(* CoDeSys 2.3 library: TcSystemCX.lib *)
(* Libraries: STANDARD.LIB 5.6.98 12:03:02, TcBase.lib*14.5.09 12:14:08, TcSystem.lib*21.1.15 10:22:54 *)

(* Global variable list: Global_Constants *)
VAR_GLOBAL CONSTANT
	iLength						 : INT := 40;
	IOADS_IGR_IODEVICESTATE_BASE : UDINT := 16#00005000;	(* plus DeviceID of CX1100 *)
END_VAR

(* Data type *)
TYPE
	E_CX1100_DisplayModes :
	(
		e_CX1100_DisplayNoAction := 0,
		e_CX1100_DisplayOn		:= 1,
		e_CX1100_DisplayOff,
		e_CX1100_CursorOn,
		e_CX1100_CursorOff,
		e_CX1100_CursorBlinkOn,
		e_CX1100_CursorBlinkOff,
		e_CX1100_BackLightOn,
		e_CX1100_BackLightOff,
		e_CX1100_ClearDisplay,
		e_CX1100_WriteLine1,
		e_CX1100_WriteLine2
	);
END_TYPE

(* Data type *)
TYPE E_CX1100_NaviSwitch : (
	e_CX1100_NaviSwitch_IDLE 			:= 0,
	e_CX1100_NaviSwitch_MIDDLE			:= 16,

	(* clockwise in 45 degree steps *)
	e_CX1100_NaviSwitch_TOP 			:= 1,
	e_CX1100_NaviSwitch_TOPRIGHT 		:= 9,
	e_CX1100_NaviSwitch_RIGHT			:= 8,
	e_CX1100_NaviSwitch_BOTTOMRIGHT		:= 10,
	e_CX1100_NaviSwitch_BOTTOM			:= 2,
	e_CX1100_NaviSwitch_BOTTOMLEFT		:= 6,
	e_CX1100_NaviSwitch_LEFT 			:= 4,
	e_CX1100_NaviSwitch_TOPLEFT 		:= 5,

	(* clockwise in 45 degree steps with middle switch pressed *)
	e_CX1100_NaviSwitch_MIDDLE_TOP 			:= 17,
	e_CX1100_NaviSwitch_MIDDLE_TOPRIGHT 	:= 25,
	e_CX1100_NaviSwitch_MIDDLE_RIGHT		:= 24,
	e_CX1100_NaviSwitch_MIDDLE_BOTTOMRIGHT	:= 26,
	e_CX1100_NaviSwitch_MIDDLE_BOTTOM		:= 18,
	e_CX1100_NaviSwitch_MIDDLE_BOTTOMLEFT	:= 22,
	e_CX1100_NaviSwitch_MIDDLE_LEFT 		:= 20,
	e_CX1100_NaviSwitch_MIDDLE_TOPLEFT 		:= 21
);
END_TYPE

(* Data type *)
TYPE
	E_CX2100_DisplayModesRd :
	(
		eCX2100_DisplayNoActionRd 	:= 0,
		eCX2100_ReadCursorInfo		:= 20,
		eCX2100_ReadBackLight,
		eCX2100_ReadLine1,
		eCX2100_ReadLine2,
		eCX2100_ReadLines
	);
END_TYPE

(* Data type *)
TYPE
	E_CX2100_DisplayModesWr :
	(
		eCX2100_DisplayNoActionWr 	:= 0,
		eCX2100_CursorOn 			:= 3,
		eCX2100_CursorOff,
		eCX2100_CursorBlinkOn,
		eCX2100_CursorBlinkOff,
		eCX2100_BackLightOn,
		eCX2100_BackLightOff,
		eCX2100_ClearDisplay,
		eCX2100_WriteLine1,
		eCX2100_WriteLine2,
		eCX2100_WriteLines,
		eCX2100_CursorPosX,
		eCX2100_CursorPosY,
		eCX2100_CursorPosXY
	);
END_TYPE

(* Data type *)
TYPE E_CX2100_NaviSwitch : (
	eCX2100_NaviSwitch_IDLE 		:= 0,
	eCX2100_NaviSwitch_MIDDLE		:= 15,
	eCX2100_NaviSwitch_ENTER		:= 16,
	eCX2100_NaviSwitch_ENTER_MIDDLE	:= 31,

	(* clockwise in 45 degree steps, 1-2 switches on *)
	eCX2100_NaviSwitch_TOP 			:= 1,
	eCX2100_NaviSwitch_TOPRIGHT 	:= 9,
	eCX2100_NaviSwitch_RIGHT		:= 8,
	eCX2100_NaviSwitch_BOTTOMRIGHT	:= 10,
	eCX2100_NaviSwitch_BOTTOM		:= 2,
	eCX2100_NaviSwitch_BOTTOMLEFT	:= 6,
	eCX2100_NaviSwitch_LEFT 		:= 4,
	eCX2100_NaviSwitch_TOPLEFT 		:= 5,

	(* clockwise in 90 degree steps, 3 switches on *)
	eCX2100_NaviSwitch_TOPLEFTRIGHT 	:= 13,
	eCX2100_NaviSwitch_RIGHTTOPBOTTOM 	:= 11,
	eCX2100_NaviSwitch_BOTTOMLEFTRIGHT	:= 14,
	eCX2100_NaviSwitch_LEFTTOPBOTTOM	:= 7,

	(* clockwise in 45 degree steps with enter switch pressed, 1-2 switches on *)
	eCX2100_NaviSwitch_ENTER_TOP 		:= 17,
	eCX2100_NaviSwitch_ENTER_TOPRIGHT 	:= 25,
	eCX2100_NaviSwitch_ENTER_RIGHT		:= 24,
	eCX2100_NaviSwitch_ENTER_BOTTOMRIGHT:= 26,
	eCX2100_NaviSwitch_ENTER_BOTTOM		:= 18,
	eCX2100_NaviSwitch_ENTER_BOTTOMLEFT	:= 22,
	eCX2100_NaviSwitch_ENTER_LEFT 		:= 20,
	eCX2100_NaviSwitch_ENTER_TOPLEFT 	:= 21,

	(* clockwise in 90 degree steps, with enter switch pressed, 3 switches on *)
	eCX2100_NaviSwitch_ENTER_TOPLEFTRIGHT 	:= 29,
	eCX2100_NaviSwitch_ENTER_RIGHTTOPBOTTOM := 27,
	eCX2100_NaviSwitch_ENTER_BOTTOMLEFTRIGHT:= 30,
	eCX2100_NaviSwitch_ENTER_LEFTTOPBOTTOM	:= 23
);
END_TYPE

(* Data type *)
TYPE E_UPS_STATE : (
	eUPS_UNDEF,
	eUPS_CHARGING,
	eUPS_CHARGED,
	eUPS_DISCHARGE,
	eUPS_DISCHARGE_RESTART,
	eUPS_OUTPUT_OFF,
	eUPS_OVERLOAD
);
END_TYPE

(* Data type *)
TYPE ST_CX_ProfilerStruct :
STRUCT
	dwLastExecTime		: DWORD;
	dwMinExecTime		: DWORD;
	dwMaxExecTime		: DWORD;
	dwAverageExecTime	: DWORD;
	dwMeasureCycle		: DWORD;
END_STRUCT
END_TYPE

(* Data type *)
TYPE ST_CxDeviceIdentification :
STRUCT
	strTargetType		: STRING(20);
	strHardwareModel	: STRING(10);
	strHardwareSerialNo	: STRING(12);
	strHardwareVersion	: STRING(4);
	strHardwareDate		: STRING(10);
	strHardwareCPU		: STRING(10);

	strImageDevice		: STRING(20);
	strImageVersion		: STRING(10);
	strImageLevel		: STRING(10);
	strImageOsName		: STRING(20);
	strImageOsVersion	: STRING(8);

	strTwinCATVersion	: STRING(4);
	strTwinCATRevision	: STRING(4);
	strTwinCATBuild		: STRING(8);
	strTwinCATLevel		: STRING(20);
	strAmsNetId			: STRING(23);
END_STRUCT
END_TYPE

(* Data type *)
TYPE ST_CxDeviceIdentificationEx :
STRUCT
	strTargetType		: STRING(30);
	strHardwareModel	: STRING(16);
	strHardwareSerialNo	: STRING(16);
	strHardwareVersion	: STRING(8);
	strHardwareDate		: STRING(12);
	strHardwareCPU		: STRING(20);

	strImageDevice		: STRING(48);
	strImageVersion		: STRING(32);
	strImageLevel		: STRING(32);
	strImageOsName		: STRING(48);
	strImageOsVersion	: STRING(8);

	strTwinCATVersion	: STRING(4);
	strTwinCATRevision	: STRING(4);
	strTwinCATBuild		: STRING(8);
	strTwinCATLevel		: STRING(20);
	strAmsNetId			: T_AmsNetId;
END_STRUCT
END_TYPE

(* POU F_CXNaviSwitch, ST *)
FUNCTION F_CXNaviSwitch : E_CX1100_NaviSwitch
VAR_INPUT
	iCX1100_IN : USINT;
END_VAR
VAR
END_VAR
F_CXNaviSwitch := USINT_TO_BYTE(iCX1100_IN) AND 16#1F;
END_FUNCTION

(* POU F_CXNaviSwitchUSB, ST *)
FUNCTION F_CXNaviSwitchUSB : E_CX2100_NaviSwitch
VAR_INPUT
	iCX2100_IN : USINT;
END_VAR
VAR
END_VAR
F_CXNaviSwitchUSB := SHR(USINT_TO_BYTE(iCX2100_IN) AND 16#7C, 2);
END_FUNCTION

(* POU F_CXSubTimeStamp, ST *)
(* Calculates "TimeStamp_A" minus "TimeStamp_B" and returns the resulting time difference
		as "F_CXSubTimeStamp" in microseconds 

 IN:	TimeStamp_A		(2 x UDINT)		[100*ns]										
		TimeStamp_B		(2 x UDINT)		[100*ns]										

 OUT:	TimeDifference	(1 x UDINT)	[us] limited to 0..4294967295us (16#FFFFFFFF)	
		negative and huge differences are returned as 4294967295us (71m34s967ms295us)	
		in case of negative or huge differences use UInt64Sub64() of TcUtilities.lib 	*)

FUNCTION F_CXSubTimeStamp : UDINT		(* [us] *)
VAR_INPUT
	nTimeStampLoDW_A	: UDINT;	(* 2*32 bit time stamp A: low DWORD					*)
	nTimeStampHiDW_A	: UDINT;	(* 2*32 bit time stamp A: high DWORD				*)
	nTimeStampLoDW_B	: UDINT;	(* 2*32 bit time stamp B: low DWORD					*)
	nTimeStampHiDW_B	: UDINT;	(* 2*32 bit time stamp B: high DWORD				*)
END_VAR
VAR
	nDeltaTimeStampLoDW	: UDINT;	(* 2*32 bit delta time stamp for low DWORD			*)
	nDeltaTimeStampHiDW	: UDINT;	(* 2*32 bit delta time stamp for high DWORD			*)
END_VAR
VAR CONSTANT
	fSCALE_LOWDW		: LREAL	:= 0.1;	(* time stamp in [100*ns]: 1=0.1 us (1.0 / 10.0)*)
	fSCALE_HIGHDW		: LREAL := 429496729.6;	(* 4294967296(2^32) / 10				*)
END_VAR
(* calculate time difference per UDINT *)
nDeltaTimeStampLoDW := nTimeStampLoDW_A - nTimeStampLoDW_B;
nDeltaTimeStampHiDW := nTimeStampHiDW_A - nTimeStampHiDW_B;

IF ( nTimeStampLoDW_A >= nTimeStampLoDW_B ) THEN
	F_CXSubTimeStamp	:= LREAL_TO_UDINT(
		LIMIT(
			0,
			UDINT_TO_LREAL(nDeltaTimeStampHiDW) * 429496729.6 + UDINT_TO_LREAL(nDeltaTimeStampLoDW) / 10.0,
			4294967295)
	);
ELSE
	F_CXSubTimeStamp	:= LREAL_TO_UDINT(
		LIMIT(
			0,
			UDINT_TO_LREAL(nDeltaTimeStampHiDW - 1) * 429496729.6 + UDINT_TO_LREAL(nDeltaTimeStampLoDW) / 10.0,
			4294967295)
	);
END_IF;
END_FUNCTION

(* POU F_GetVersionTcSystemCX, ST *)
FUNCTION F_GetVersionTcSystemCX : UINT
VAR_INPUT
	nVersionElement		:	INT;
END_VAR
(*
	Possible nVersionElement parameter:
	1	:	major number
	2	:	minor number
	3	:	revision number
*)
VAR
END_VAR
(* For embedded controllers of the CX series use:
   - for the CX1000 the generic TcSystemCX.lib + the TcSystemCX1000.lib 
     (the TcCX1000System.lib is discontinued, should not be used in new projects)

   - for the CX1010 the generic TcSystemCX.lib + the TcSystemCX1010.lib
   - for the CX1020 the generic TcSystemCX.lib + the TcSystemCX1020.lib
   - for the CX1030 the generic TcSystemCX.lib + the TcSystemCX1030.lib
   - for the CX5010 the generic TcSystemCX.lib + the TcSystemCX5010.lib
   - for the CX5020 the generic TcSystemCX.lib + the TcSystemCX5020.lib
   - for the CX9000 the generic TcSystemCX.lib + the TcSystemCX9000.lib
   - for the CX9010 the generic TcSystemCX.lib + the TcSystemCX9010.lib

   - ...
*)

(* Version history:
Date         	| Version    	| created under      				| Author          		| Remark 
--------------------------------------------------------------------------------------------------------------------------------------------------------------------- 
2006/02/28    	| 1.1.0      	| V2.10.0 (Build 1247)				| ICh		    		| created from TcCX1000System.lib v1.0.2
2006/03/02    	| 1.1.1      	| V2.10.0 (Build 1247)				| ICh		    		| F_CX_NaviSwitch + E_CX1100_NaviSwitch added
2006/03/02    	| 1.1.2      	| V2.10.0 (Build 1247)				| ICh		    		| E_CX1100_NaviSwitch extended
2006/04/11    	| 1.1.3      	| V2.10.0 (Build 1255)				| ICh		    		| change to FB_CXSimpleUps (added check that input links exist)
2006/08/10    	| 1.1.4      	| V2.10.0 (Build 1302)				| ICh		    		| FB_CXSimpleUps avoids possible deadlock (Win and Tc Stopped, CX Power supply running)
2006/08/10    	| 1.1.5      	| V2.10.0 (Build 1302)				| ICh		    		| FB_CxGetDeviceIdentification added
2006/08/19    	| 1.1.6      	| V2.10.0 (Build 1302)				| ICh		    		| reduced realtim load of FB_CxGetDeviceIdentification
2007/01/29    	| 1.1.7      	| V2.10.0 (Build 1307)				| ICh		    		| fix for F_CXSubTimeStamp for larger/negative differences
2007/02/16    	| 1.1.8      	| V2.10.0 (Build 1309)				| ICh		    		| saved as internal 2.10 lib
2007/03/05    	| 1.1.9      	| V2.10.0 (Build 1309)				| ICh		    		| added CPU-Architecture to FB_CxGetDeviceIdentification
2007/03/05    	| 1.1.10      	| V2.10.0 (Build 1319)				| ICh		    		| FB_CXSimpleUps extended internal holding, always holding until time ellapsed, 
																								limiting UPS holding time between 0.5 and 10s
2007/03/05    	| 1.1.11      	| V2.10.0 (Build 1319)				| ICh		    		| FB_CXSimpleUps fix for power off
2007/03/05    	| 1.1.12      	| V2.10.0 (Build 1319)				| ICh		    		| FB_CXSimpleUps cleanup
2007/03/05    	| 1.1.13      	| V2.10.0 (Build 1319)				| ICh		    		| FB_CXSimpleUps optimization
2007/10/06    	| 1.1.14      	| V2.10.0 (Build 1319)				| ICh		    		| Fix for CursorOff in FB_CXSetTextDisplay
11.10.2010	| 1.1.15	|	TCAT2.11 B2015				|	Christoph C	| Small correction in the FB_CXProfiler function block (calculation of average velue for a first measure cycle )
24.01.2011	| 1.1.16	|	TCAT2.11 B2021				|	I.Ch.	| limiting string copy operations in FB_CxGetDeviceIdentification
08.02.2012	| 1.1.17	|	TCAT2.11 B2217				|	I.Ch.	| added FB_CxGetDeviceIdentificationEx
17.06.2013	| 1.1.18	|	TCAT2.11 B2234				|	I.Ch.	| added FB_CXGetTextDisplayUSB, FB_CXSetTextDisplayUSB, F_CXNaviSwitchUSB and corresponding DTs for CX2100 display + navi switch
06.12.2013	| 1.1.19	|	TCAT2.11 B2239				|	I.Ch.	| added small adjustements to FB_CXGetTextDisplayUSB, FB_CXSetTextDisplayUSB in order to be used with EL6080 too
07.09.2016	| 1.1.20	|	TCAT2.11 B2254				|	I.Ch.	| change type from INT to UDINT due to signed/unsigned warning in FB_CXProfiler
*) 
CASE nVersionElement OF
1:	(* major number *)
	F_GetVersionTcSystemCX := 1;
2:	(* minor number *)
	F_GetVersionTcSystemCX := 1;
3:	(* revision number *)
	F_GetVersionTcSystemCX := 20;
ELSE
	F_GetVersionTcSystemCX := 16#FFFF;
END_CASE
END_FUNCTION

(* POU FB_CxGetDeviceIdentification, ST *)
FUNCTION_BLOCK FB_CxGetDeviceIdentification
VAR_INPUT
	bExecute 		: BOOL;
	tTimeout		: TIME;
END_VAR
VAR_OUTPUT
	bBusy 			: BOOL;
	bError			: BOOL;
	nErrorID		: UDINT;
	stDevIdent 		: ST_CxDeviceIdentification;
END_VAR
VAR CONSTANT
	iDataSize		: INT  := 1024;
	byTagStart		: BYTE := 60; (* '<' *)
	byTagEnd		: BYTE := 62; (* '>' *)
	byTagSlash		: BYTE := 47; (* '/' *)
END_VAR
VAR
	fbAdsRead		: ADSREAD;
	bExecutePrev	: BOOL;
	iState			: INT;
	iData			: ARRAY [1..iDataSize] OF BYTE;
	strActPath		: STRING(255);
	iLoopEndIdx		: INT;
	iStructSize		: UDINT;
	strHardwareCPU	: STRING(10);

	strTags			: ARRAY [0..9] OF STRING(40);
	iTagsSize		: ARRAY [0..9] OF UDINT;
	iCurrTag		: ARRAY [0..40] OF BYTE;
	iCurrTagData	: ARRAY [0..80] OF BYTE;
	iPathSize		: UDINT;

	iTagIdx			: INT;
	iCurrTagIdx		: INT;
	iDataIdx		: INT;
	iCurrTagDataIdx	: INT;
	k				: INT;
	iMinCurrData	: INT;
	iFirstIdx		: INT;
	iLastIdx		: INT;

	bTagStart		: BOOL;
	bTagEnd			: BOOL;
	bTagSlash		: BOOL;
	bTagOpen		: BOOL;
END_VAR
CASE iState OF
0: (* IDLE *)
	IF bExecute AND NOT bExecutePrev THEN
		bExecutePrev 	:= TRUE;
		bBusy 			:= TRUE;
		bError			:= FALSE;
		nErrorID		:= 0;
		iStructSize 	:= SIZEOF(stDevIdent);
		strActPath		:= '';
		iCurrTagIdx		:= 0;
		iTagIdx			:= 0;
		bTagStart		:= FALSE;
		bTagEnd			:= FALSE;
		bTagSlash		:= FALSE;
		bTagOpen		:= FALSE;
		iMinCurrData	:= 0;
		iDataIdx		:= 0;
		iLoopEndIdx		:= 0;
		iFirstIdx 		:= 0;
		iLastIdx 		:= 0;
		iPathSize		:= 0;

		MEMSET(ADR(iData), 0, SIZEOF(iData));
		MEMSET(ADR(stDevIdent), 0, SIZEOF(stDevIdent));
		MEMSET(ADR(iCurrTag), 0, SIZEOF(iCurrTag));
		MEMSET(ADR(iCurrTagData), 0, SIZEOF(iCurrTagData));
		MEMSET(ADR(iTagsSize), 0, SIZEOF(iTagsSize));

		(* get device identification *)
		fbAdsRead(
			NETID	:= '',
			PORT	:= 10000,
			IDXGRP	:= 700,
			IDXOFFS	:= 1,
			LEN		:= SIZEOF(iData),
			DESTADDR:= ADR(iData),
			READ	:= FALSE,
			TMOUT	:= T#3s
		);
		fbAdsRead(READ := TRUE);

		iState := 1;
	END_IF

1: (* wait for read done *)
	fbAdsRead();

	IF NOT fbAdsRead.BUSY THEN
		bError	 := fbAdsRead.ERR;
		nErrorID := fbAdsRead.ERRID;

		IF fbAdsRead.ERR THEN
			fbAdsRead(READ := FALSE);
			iState := 0;
			bBusy  := FALSE;
		ELSE
			fbAdsRead(READ := FALSE);
			iLoopEndIdx := MIN(UDINT_TO_INT(fbAdsRead.fbAdsRead.cbRead), iDataSize);
			iFirstIdx := 1;
			iLastIdx := 64;
			iState := 2;
		END_IF
	END_IF

2: (* evaluate data *)
	(* parse data for known tags and their values *)
	iFirstIdx := MIN(iFirstIdx, iLoopEndIdx);
	iLastIdx := MIN(iLastIdx, iLoopEndIdx);

	FOR iDataIdx := iFirstIdx TO iLastIdx DO
		IF NOT bTagStart AND NOT bTagEnd AND (iData[iDataIdx] = byTagStart) THEN
			(* start of new tag '<...' *)
			bTagStart	:= TRUE;
			bTagEnd		:= FALSE;
			bTagSlash	:= FALSE;
			iCurrTagIdx	:= 0;
			iCurrTag[iCurrTagIdx] := iData[iDataIdx];
			iCurrTagIdx	:= iCurrTagIdx + 1;

		ELSIF bTagStart AND (iData[iDataIdx] = byTagSlash) THEN
			(* this is a closing tag '</...' *)
			bTagSlash	:= TRUE;
			iCurrTag[iCurrTagIdx] := iData[iDataIdx];
			iCurrTagIdx	:= iCurrTagIdx + 1;

		ELSIF bTagStart AND NOT bTagEnd AND iData[iDataIdx] = byTagEnd THEN
			(* end of new tag '...>' *)
			bTagStart	:= FALSE;
			bTagEnd		:= TRUE;
			iCurrTag[iCurrTagIdx] := iData[iDataIdx];
			iCurrTagIdx	:= iCurrTagIdx + 1;

			(* end of closing tag '</xyz>' - evaluate tag data *)
			IF bTagSlash THEN
				(* remove level *)
				iTagIdx := MAX(iTagIdx - 1, 0);
				MEMSET(ADR(strTags[iTagIdx]), 0, SIZEOF(strTags[iTagIdx]));

				(* get current tag data *)
				IF iCurrTagDataIdx > 0 THEN
					iMinCurrData := MIN(SIZEOF(iCurrTagData), iCurrTagDataIdx);

					(* assign data to structure if corresponding tag was found *)
					IF strActPath = '<TcTargetDesc><TargetType>' THEN
						MEMCPY(ADR(stDevIdent.strTargetType), 		ADR(iCurrTagData),
							MIN(SIZEOF(stDevIdent.strTargetType)-1, iMinCurrData));

					ELSIF strActPath = '<TcTargetDesc><TargetVersion><Version>' THEN
						MEMCPY(ADR(stDevIdent.strTwinCATVersion), 	ADR(iCurrTagData),
							MIN(SIZEOF(stDevIdent.strTwinCATVersion)-1, iMinCurrData));

					ELSIF strActPath = '<TcTargetDesc><TargetVersion><Revision>' THEN
						MEMCPY(ADR(stDevIdent.strTwinCATRevision), 	ADR(iCurrTagData),
							MIN(SIZEOF(stDevIdent.strTwinCATRevision)-1, iMinCurrData));

					ELSIF strActPath = '<TcTargetDesc><TargetVersion><Build>' THEN
						MEMCPY(ADR(stDevIdent.strTwinCATBuild), 	ADR(iCurrTagData),
							MIN(SIZEOF(stDevIdent.strTwinCATBuild)-1, iMinCurrData));

					ELSIF strActPath = '<TcTargetDesc><TargetFeatures><Level>' THEN
						MEMCPY(ADR(stDevIdent.strTwinCATLevel), 	ADR(iCurrTagData),
							MIN(SIZEOF(stDevIdent.strTwinCATLevel)-1, iMinCurrData));

					ELSIF strActPath = '<TcTargetDesc><TargetFeatures><NetId>' THEN
						MEMCPY(ADR(stDevIdent.strAmsNetId), 		ADR(iCurrTagData),
							MIN(SIZEOF(stDevIdent.strAmsNetId)-1, iMinCurrData));

					ELSIF strActPath = '<TcTargetDesc><Hardware><Model>' THEN
						MEMCPY(ADR(stDevIdent.strHardwareModel), 	ADR(iCurrTagData),
							MIN(SIZEOF(stDevIdent.strHardwareModel)-1, iMinCurrData));

					ELSIF strActPath = '<TcTargetDesc><Hardware><SerialNo>' THEN
						MEMCPY(ADR(stDevIdent.strHardwareSerialNo), ADR(iCurrTagData),
							MIN(SIZEOF(stDevIdent.strHardwareSerialNo)-1, iMinCurrData));

					ELSIF strActPath = '<TcTargetDesc><Hardware><CPUVersion>' THEN
						MEMCPY(ADR(stDevIdent.strHardwareVersion), 	ADR(iCurrTagData),
							MIN(SIZEOF(stDevIdent.strHardwareVersion)-1, iMinCurrData));

					ELSIF strActPath = '<TcTargetDesc><Hardware><Date>' THEN
						MEMCPY(ADR(stDevIdent.strHardwareDate), 	ADR(iCurrTagData),
							MIN(SIZEOF(stDevIdent.strHardwareDate)-1, iMinCurrData));

					ELSIF strActPath = '<TcTargetDesc><Hardware><CPUArchitecture>' THEN
						MEMCPY(ADR(strHardwareCPU), ADR(iCurrTagData),
							MIN(SIZEOF(strHardwareCPU)-1, iMinCurrData));

						IF strHardwareCPU = '0' THEN
							stDevIdent.strHardwareCPU := 'INTELx86';
						ELSIF strHardwareCPU = '1' THEN
							stDevIdent.strHardwareCPU := 'MIPS';
						ELSIF strHardwareCPU = '2' THEN
							stDevIdent.strHardwareCPU := 'ALPHA';
						ELSIF strHardwareCPU = '3' THEN
							stDevIdent.strHardwareCPU := 'PPC';
						ELSIF strHardwareCPU = '4' THEN
							stDevIdent.strHardwareCPU := 'SHX';
						ELSIF strHardwareCPU = '5' THEN
							stDevIdent.strHardwareCPU := 'ARM';
						ELSIF strHardwareCPU = '6' THEN
							stDevIdent.strHardwareCPU := 'IA64';
						ELSIF strHardwareCPU = '7' THEN
							stDevIdent.strHardwareCPU := 'ALPHA64';
						ELSIF strHardwareCPU = '8' THEN
							stDevIdent.strHardwareCPU := 'MSIL';
						ELSIF strHardwareCPU = '9' THEN
							stDevIdent.strHardwareCPU := 'AMDx64';
						ELSIF strHardwareCPU = '10' THEN
							stDevIdent.strHardwareCPU := 'IA32_ON_WIN64';
						ELSE
							stDevIdent.strHardwareCPU := 'UNKNOWN';
						END_IF
						strHardwareCPU := '';

					ELSIF strActPath = '<TcTargetDesc><OsImage><ImageDevice>' THEN
						MEMCPY(ADR(stDevIdent.strImageDevice), 		ADR(iCurrTagData),
							MIN(SIZEOF(stDevIdent.strImageDevice)-1, iMinCurrData));

					ELSIF strActPath = '<TcTargetDesc><OsImage><ImageVersion>' THEN
						MEMCPY(ADR(stDevIdent.strImageVersion), 	ADR(iCurrTagData),
							MIN(SIZEOF(stDevIdent.strImageVersion)-1, iMinCurrData));

					ELSIF strActPath = '<TcTargetDesc><OsImage><ImageLevel>' THEN
						MEMCPY(ADR(stDevIdent.strImageLevel), 		ADR(iCurrTagData),
							MIN(SIZEOF(stDevIdent.strImageLevel)-1, iMinCurrData));

					ELSIF strActPath = '<TcTargetDesc><OsImage><OsName>' THEN
						MEMCPY(ADR(stDevIdent.strImageOsName), 		ADR(iCurrTagData),
							MIN(SIZEOF(stDevIdent.strImageOsName)-1, iMinCurrData));

					ELSIF strActPath = '<TcTargetDesc><OsImage><OsVersion>' THEN
						MEMCPY(ADR(stDevIdent.strImageOsVersion), 	ADR(iCurrTagData),
							MIN(SIZEOF(stDevIdent.strImageOsVersion)-1, iMinCurrData));
					END_IF

					iCurrTagDataIdx	:= 0;
				END_IF

				bTagOpen := FALSE;
			ELSE
				(* add level with current tag *)
				iTagsSize[iTagIdx] := MIN(MIN(SIZEOF(strTags[iTagIdx]), SIZEOF(iCurrTag)), iCurrTagIdx);

				MEMSET(ADR(strTags[iTagIdx]), 0, SIZEOF(strTags[iTagIdx]));
				MEMCPY(ADR(strTags[iTagIdx]), ADR(iCurrTag), iTagsSize[iTagIdx]);
				MEMSET(ADR(strActPath), 0, SIZEOF(strActPath));
				iPathSize	:= 0;

				FOR k := 0 TO iTagIdx DO
					MEMCPY(ADR(strActPath) + iPathSize, ADR(strTags[k]), iTagsSize[k]);
					iPathSize := iPathSize + iTagsSize[k];
				END_FOR

				iTagIdx := MIN(iTagIdx + 1, 9);

				bTagOpen := TRUE;
			END_IF

			bTagEnd := FALSE;
		ELSIF bTagStart THEN
			(* receiving new tag '<...xyz...>' or '</...xyz...>' *)
			iCurrTag[iCurrTagIdx] := iData[iDataIdx];
			iCurrTagIdx	:= iCurrTagIdx + 1;

		ELSIF bTagOpen THEN
			(* receiving new data '<xyz>...nnn...</xyz>' *)
			iCurrTagData[iCurrTagDataIdx] := iData[iDataIdx];
			iCurrTagDataIdx	:= iCurrTagDataIdx + 1;

		END_IF
	END_FOR

	iFirstIdx := iFirstIdx + 64;
	iLastIdx := iLastIdx + 64;

	IF iFirstIdx > iLoopEndIdx THEN
		iState := 3;
	END_IF

3: (* cleanup *)
	MEMSET(ADR(iData), 0, SIZEOF(iData));
	MEMSET(ADR(iCurrTag), 0, SIZEOF(iCurrTag));
	MEMSET(ADR(iCurrTagData), 0, SIZEOF(iCurrTagData));
	MEMSET(ADR(iTagsSize), 0, SIZEOF(iTagsSize));

	strActPath		:= '';
	iCurrTagIdx		:= 0;
	iTagIdx			:= 0;
	bTagStart		:= FALSE;
	bTagEnd			:= FALSE;
	bTagSlash		:= FALSE;
	bTagOpen		:= FALSE;
	iMinCurrData	:= 0;
	iDataIdx		:= 0;
	iLoopEndIdx		:= 0;
	iFirstIdx 		:= 0;
	iLastIdx 		:= 0;
	iPathSize		:= 0;

	iState 			:= 0;
	bBusy 			:= FALSE;

END_CASE

(* auto clear *)
bExecutePrev := bExecutePrev AND bExecute;
END_FUNCTION_BLOCK

(* POU FB_CxGetDeviceIdentificationEx, ST *)
FUNCTION_BLOCK FB_CxGetDeviceIdentificationEx
VAR_INPUT
	bExecute 		: BOOL;(* Rising edge on this input activates the fb execution *)
	tTimeout		: TIME := DEFAULT_ADS_TIMEOUT;
	sNetId			: T_AmsNetId;	(* Ams net id of target system *)
END_VAR
VAR_OUTPUT
	bBusy 			: BOOL;
	bError			: BOOL;
	nErrorID		: UDINT;
	stDevIdent 		: ST_CxDeviceIdentificationEx;(* structure with available device identification data *)
END_VAR
{library private}
VAR CONSTANT
	iDataSize		: INT  := 2048;
	byTagStart		: BYTE := 60; (* '<' *)
	byTagEnd		: BYTE := 62; (* '>' *)
	byTagSlash	: BYTE := 47; (* '/' *)
END_VAR
VAR
	fbAdsRead		: ADSREAD;
	bExecutePrev	: BOOL;
	iState			: INT;
	iData			: ARRAY [1..iDataSize] OF BYTE;
	strActPath		: STRING(255);
	iLoopEndIdx		: INT;
	iStructSize		: UDINT;
	strHardwareCPU	: STRING(10);

	strTags			: ARRAY [0..9] OF STRING(40);
	iTagsSize		: ARRAY [0..9] OF UDINT;
	iCurrTag		: ARRAY [0..40] OF BYTE;
	iCurrTagData	: ARRAY [0..80] OF BYTE;
	iPathSize		: UDINT;

	iTagIdx			: INT;
	iCurrTagIdx		: INT;
	iDataIdx		: INT;
	iCurrTagDataIdx	: INT;
	k				: INT;
	iMinCurrData	: INT;
	iFirstIdx		: INT;
	iLastIdx		: INT;

	bTagStart		: BOOL;
	bTagEnd			: BOOL;
	bTagSlash		: BOOL;
	bTagOpen		: BOOL;
END_VAR
CASE iState OF
0: (* IDLE *)
	IF bExecute AND NOT bExecutePrev THEN
		bExecutePrev 	:= TRUE;
		bBusy 			:= TRUE;
		bError			:= FALSE;
		nErrorID		:= 0;
		iStructSize 	:= SIZEOF(stDevIdent);
		strActPath		:= '';
		iCurrTagIdx		:= 0;
		iTagIdx			:= 0;
		bTagStart		:= FALSE;
		bTagEnd			:= FALSE;
		bTagSlash		:= FALSE;
		bTagOpen		:= FALSE;
		iMinCurrData	:= 0;
		iDataIdx		:= 0;
		iLoopEndIdx		:= 0;
		iFirstIdx 		:= 0;
		iLastIdx 		:= 0;
		iPathSize		:= 0;

		MEMSET(ADR(iData), 0, SIZEOF(iData));
		MEMSET(ADR(stDevIdent), 0, SIZEOF(stDevIdent));
		MEMSET(ADR(iCurrTag), 0, SIZEOF(iCurrTag));
		MEMSET(ADR(iCurrTagData), 0, SIZEOF(iCurrTagData));
		MEMSET(ADR(iTagsSize), 0, SIZEOF(iTagsSize));

		(* get device identification *)
		fbAdsRead(
			NETID	:= sNetId,
			PORT	:= 10000,
			IDXGRP	:= 700,
			IDXOFFS	:= 1,
			LEN		:= SIZEOF(iData),
			DESTADDR:= ADR(iData),
			READ	:= FALSE,
			TMOUT	:= T#3s
		);
		fbAdsRead(READ := TRUE);

		iState := 1;
	END_IF

1: (* wait for read done *)
	fbAdsRead();

	IF NOT fbAdsRead.BUSY THEN
		bError	 := fbAdsRead.ERR;
		nErrorID := fbAdsRead.ERRID;

		IF fbAdsRead.ERR THEN
			fbAdsRead(READ := FALSE);
			iState := 0;
			bBusy  := FALSE;
		ELSE
			fbAdsRead(READ := FALSE);
			iLoopEndIdx := MIN(UDINT_TO_INT(fbAdsRead.fbAdsRead.cbRead), iDataSize);
			iFirstIdx := 1;
			iLastIdx := 64;
			iState := 2;
		END_IF
	END_IF

2: (* evaluate data *)
	(* parse data for known tags and their values *)
	iFirstIdx := MIN(iFirstIdx, iLoopEndIdx);
	iLastIdx := MIN(iLastIdx, iLoopEndIdx);

	FOR iDataIdx := iFirstIdx TO iLastIdx DO
		IF NOT bTagStart AND NOT bTagEnd AND (iData[iDataIdx] = byTagStart) THEN
			(* start of new tag '<...' *)
			bTagStart	:= TRUE;
			bTagEnd		:= FALSE;
			bTagSlash	:= FALSE;
			iCurrTagIdx	:= 0;
			iCurrTag[iCurrTagIdx] := iData[iDataIdx];
			iCurrTagIdx	:= iCurrTagIdx + 1;

		ELSIF bTagStart AND (iData[iDataIdx] = byTagSlash) THEN
			(* this is a closing tag '</...' *)
			bTagSlash	:= TRUE;
			iCurrTag[iCurrTagIdx] := iData[iDataIdx];
			iCurrTagIdx	:= iCurrTagIdx + 1;

		ELSIF bTagStart AND NOT bTagEnd AND iData[iDataIdx] = byTagEnd THEN
			(* end of new tag '...>' *)
			bTagStart	:= FALSE;
			bTagEnd		:= TRUE;
			iCurrTag[iCurrTagIdx] := iData[iDataIdx];
			iCurrTagIdx	:= iCurrTagIdx + 1;

			(* end of closing tag '</xyz>' - evaluate tag data *)
			IF bTagSlash THEN
				(* remove level *)
				iTagIdx := MAX(iTagIdx - 1, 0);
				MEMSET(ADR(strTags[iTagIdx]), 0, SIZEOF(strTags[iTagIdx]));

				(* get current tag data *)
				IF iCurrTagDataIdx > 0 THEN
					iMinCurrData := MIN(SIZEOF(iCurrTagData), iCurrTagDataIdx);

					(* assign data to structure if corresponding tag was found *)
					IF strActPath = '<TcTargetDesc><TargetType>' THEN
						MEMCPY(ADR(stDevIdent.strTargetType), 		ADR(iCurrTagData),
							MIN(SIZEOF(stDevIdent.strTargetType)-1, iMinCurrData));

					ELSIF strActPath = '<TcTargetDesc><TargetVersion><Version>' THEN
						MEMCPY(ADR(stDevIdent.strTwinCATVersion), 	ADR(iCurrTagData),
							MIN(SIZEOF(stDevIdent.strTwinCATVersion)-1, iMinCurrData));

					ELSIF strActPath = '<TcTargetDesc><TargetVersion><Revision>' THEN
						MEMCPY(ADR(stDevIdent.strTwinCATRevision), 	ADR(iCurrTagData),
							MIN(SIZEOF(stDevIdent.strTwinCATRevision)-1, iMinCurrData));

					ELSIF strActPath = '<TcTargetDesc><TargetVersion><Build>' THEN
						MEMCPY(ADR(stDevIdent.strTwinCATBuild), 	ADR(iCurrTagData),
							MIN(SIZEOF(stDevIdent.strTwinCATBuild)-1, iMinCurrData));

					ELSIF strActPath = '<TcTargetDesc><TargetFeatures><Level>' THEN
						MEMCPY(ADR(stDevIdent.strTwinCATLevel), 	ADR(iCurrTagData),
							MIN(SIZEOF(stDevIdent.strTwinCATLevel)-1, iMinCurrData));

					ELSIF strActPath = '<TcTargetDesc><TargetFeatures><NetId>' THEN
						MEMCPY(ADR(stDevIdent.strAmsNetId), 		ADR(iCurrTagData),
							MIN(SIZEOF(stDevIdent.strAmsNetId)-1, iMinCurrData));

					ELSIF strActPath = '<TcTargetDesc><Hardware><Model>' THEN
						MEMCPY(ADR(stDevIdent.strHardwareModel), 	ADR(iCurrTagData),
							MIN(SIZEOF(stDevIdent.strHardwareModel)-1, iMinCurrData));

					ELSIF strActPath = '<TcTargetDesc><Hardware><SerialNo>' THEN
						MEMCPY(ADR(stDevIdent.strHardwareSerialNo), ADR(iCurrTagData),
							MIN(SIZEOF(stDevIdent.strHardwareSerialNo)-1, iMinCurrData));

					ELSIF strActPath = '<TcTargetDesc><Hardware><CPUVersion>' THEN
						MEMCPY(ADR(stDevIdent.strHardwareVersion), 	ADR(iCurrTagData),
							MIN(SIZEOF(stDevIdent.strHardwareVersion)-1, iMinCurrData));

					ELSIF strActPath = '<TcTargetDesc><Hardware><Date>' THEN
						MEMCPY(ADR(stDevIdent.strHardwareDate), 	ADR(iCurrTagData),
							MIN(SIZEOF(stDevIdent.strHardwareDate)-1, iMinCurrData));

					ELSIF strActPath = '<TcTargetDesc><Hardware><CPUArchitecture>' THEN
						MEMCPY(ADR(strHardwareCPU), ADR(iCurrTagData),
							MIN(SIZEOF(strHardwareCPU)-1, iMinCurrData));

						IF strHardwareCPU = '0' THEN
							stDevIdent.strHardwareCPU := 'INTELx86';
						ELSIF strHardwareCPU = '1' THEN
							stDevIdent.strHardwareCPU := 'MIPS';
						ELSIF strHardwareCPU = '2' THEN
							stDevIdent.strHardwareCPU := 'ALPHA';
						ELSIF strHardwareCPU = '3' THEN
							stDevIdent.strHardwareCPU := 'PPC';
						ELSIF strHardwareCPU = '4' THEN
							stDevIdent.strHardwareCPU := 'SHX';
						ELSIF strHardwareCPU = '5' THEN
							stDevIdent.strHardwareCPU := 'ARM';
						ELSIF strHardwareCPU = '6' THEN
							stDevIdent.strHardwareCPU := 'IA64';
						ELSIF strHardwareCPU = '7' THEN
							stDevIdent.strHardwareCPU := 'ALPHA64';
						ELSIF strHardwareCPU = '8' THEN
							stDevIdent.strHardwareCPU := 'MSIL';
						ELSIF strHardwareCPU = '9' THEN
							stDevIdent.strHardwareCPU := 'AMDx64';
						ELSIF strHardwareCPU = '10' THEN
							stDevIdent.strHardwareCPU := 'IA32_ON_WIN64';
						ELSE
							stDevIdent.strHardwareCPU := 'UNKNOWN';
						END_IF
						strHardwareCPU := '';

					ELSIF strActPath = '<TcTargetDesc><OsImage><ImageDevice>' THEN
						MEMCPY(ADR(stDevIdent.strImageDevice), 		ADR(iCurrTagData),
							MIN(SIZEOF(stDevIdent.strImageDevice)-1, iMinCurrData));

					ELSIF strActPath = '<TcTargetDesc><OsImage><ImageVersion>' THEN
						MEMCPY(ADR(stDevIdent.strImageVersion), 	ADR(iCurrTagData),
							MIN(SIZEOF(stDevIdent.strImageVersion)-1, iMinCurrData));

					ELSIF strActPath = '<TcTargetDesc><OsImage><ImageLevel>' THEN
						MEMCPY(ADR(stDevIdent.strImageLevel), 		ADR(iCurrTagData),
							MIN(SIZEOF(stDevIdent.strImageLevel)-1, iMinCurrData));

					ELSIF strActPath = '<TcTargetDesc><OsImage><OsName>' THEN
						MEMCPY(ADR(stDevIdent.strImageOsName), 		ADR(iCurrTagData),
							MIN(SIZEOF(stDevIdent.strImageOsName)-1, iMinCurrData));

					ELSIF strActPath = '<TcTargetDesc><OsImage><OsVersion>' THEN
						MEMCPY(ADR(stDevIdent.strImageOsVersion), 	ADR(iCurrTagData),
							MIN(SIZEOF(stDevIdent.strImageOsVersion)-1, iMinCurrData));
					END_IF

					iCurrTagDataIdx	:= 0;
				END_IF

				bTagOpen := FALSE;
			ELSE
				(* add level with current tag *)
				iTagsSize[iTagIdx] := MIN(MIN(SIZEOF(strTags[iTagIdx]), SIZEOF(iCurrTag)), iCurrTagIdx);

				MEMSET(ADR(strTags[iTagIdx]), 0, SIZEOF(strTags[iTagIdx]));
				MEMCPY(ADR(strTags[iTagIdx]), ADR(iCurrTag), iTagsSize[iTagIdx]);
				MEMSET(ADR(strActPath), 0, SIZEOF(strActPath));
				iPathSize	:= 0;

				FOR k := 0 TO iTagIdx DO
					MEMCPY(ADR(strActPath) + iPathSize, ADR(strTags[k]), iTagsSize[k]);
					iPathSize := iPathSize + iTagsSize[k];
				END_FOR

				iTagIdx := MIN(iTagIdx + 1, 9);

				bTagOpen := TRUE;
			END_IF

			bTagEnd := FALSE;
		ELSIF bTagStart THEN
			(* receiving new tag '<...xyz...>' or '</...xyz...>' *)
			iCurrTag[iCurrTagIdx] := iData[iDataIdx];
			iCurrTagIdx	:= iCurrTagIdx + 1;

		ELSIF bTagOpen THEN
			(* receiving new data '<xyz>...nnn...</xyz>' *)
			iCurrTagData[iCurrTagDataIdx] := iData[iDataIdx];
			iCurrTagDataIdx	:= iCurrTagDataIdx + 1;

		END_IF
	END_FOR

	iFirstIdx := iFirstIdx + 64;
	iLastIdx := iLastIdx + 64;

	IF iFirstIdx > iLoopEndIdx THEN
		iState := 3;
	END_IF

3: (* cleanup *)
	MEMSET(ADR(iData), 0, SIZEOF(iData));
	MEMSET(ADR(iCurrTag), 0, SIZEOF(iCurrTag));
	MEMSET(ADR(iCurrTagData), 0, SIZEOF(iCurrTagData));
	MEMSET(ADR(iTagsSize), 0, SIZEOF(iTagsSize));

	strActPath		:= '';
	iCurrTagIdx		:= 0;
	iTagIdx			:= 0;
	bTagStart		:= FALSE;
	bTagEnd			:= FALSE;
	bTagSlash		:= FALSE;
	bTagOpen		:= FALSE;
	iMinCurrData	:= 0;
	iDataIdx		:= 0;
	iLoopEndIdx		:= 0;
	iFirstIdx 		:= 0;
	iLastIdx 		:= 0;
	iPathSize		:= 0;

	iState 			:= 0;
	bBusy 			:= FALSE;

END_CASE

(* auto clear *)
bExecutePrev := bExecutePrev AND bExecute;
END_FUNCTION_BLOCK

(* POU FB_CXGetTextDisplayUSB, ST *)
FUNCTION_BLOCK FB_CXGetTextDisplayUSB
VAR_INPUT
	bExecute		: BOOL;
	sNetID			: T_AmsNetID;
	nPort			: T_AmsPort;
	eMode			: E_CX2100_DisplayModesRd;
END_VAR
VAR_OUTPUT
	bBusy 			: BOOL;
	bError			: BOOL;
	nErrorID		: UDINT;
	sLine1 			: STRING;
	sLine2 			: STRING;
	nCursorPosX		: USINT;
	nCursorPosY		: USINT;
	nCursorMode		: USINT;
	nBacklight		: USINT;
END_VAR
{library private}
VAR
	eModeAct		: E_CX2100_DisplayModesRd;
	nState 			: INT := 0;
	bStarted 		: BOOL;
	fbOnTrigger		: R_TRIG;
	fbADSRead 		: ADSREADEX;
	nIndexOffset	: UDINT;
	nReadMode 		: INT;
	nReadState		: INT;
	nReadStateMax	: INT;
END_VAR
VAR CONSTANT
	(* read mode *)
	READ_MODE_IDLE	: INT := 1;
	READ_MODE_BYTE	: INT := 2;
	READ_MODE_STRING: INT := 3;

	(* CX2100*)
	IOADS_IOF_CX2100_BACKLIGHT_INT 	: UDINT := 16#80000011; (* backlight 0..255 *)
	IOADS_IOF_CX2100_LINE1 			: UDINT := 16#80080011; (* read/write line 1 STRING(80) *)
	IOADS_IOF_CX2100_LINE2		 	: UDINT := 16#80080012; (* read/write line 2 STRING(80) *)
	IOADS_IOF_CX2100_CURSOR		 	: UDINT := 16#80080019; (* cursor ... 0 Off; 1 On; 2 Blink *)
	IOADS_IOF_CX2100_CURSOR_XPOS 	: UDINT := 16#8008001A; (* cursor position in X 0..15 *)
	IOADS_IOF_CX2100_CURSOR_YPOS 	: UDINT := 16#8008001B; (* cursor position in Y 0..1 *)
	IOADS_IOF_IGRP					: UDINT	:= 16#F302;		(* ADS index group OF the CX2100 mailbox *)
END_VAR
{library public}
CASE nState OF
0 :
	fbOnTrigger(CLK:= bExecute);
    IF fbOnTrigger.Q OR bStarted THEN
		(* initialize command *)
		IF NOT bStarted THEN
			bBusy 			:= TRUE;
			bError 			:= FALSE;
			nErrorID 		:= 0;
			eModeAct	 	:= eMode;
			nReadState		:= 0;
			nReadStateMax	:= 0;
		END_IF

		(* select action *)
		CASE eModeAct OF
		eCX2100_DisplayNoActionRd:
			nIndexOffset := 0;
			nReadMode 	 := READ_MODE_IDLE;
		eCX2100_ReadCursorInfo:
			nReadStateMax := 3;
			IF NOT bStarted THEN
				nReadState := 1;
			END_IF
			CASE nReadState OF
			1:
				(* CursorPosX *)
				nIndexOffset 		:= IOADS_IOF_CX2100_CURSOR_XPOS;
				nReadMode	 		:= READ_MODE_BYTE;
				fbADSRead.DESTADDR 	:= ADR(nCursorPosX);
				fbADSRead.LEN		:= SIZEOF(nCursorPosX);
			2:
				(* CursorPosY *)
				nIndexOffset 		:= IOADS_IOF_CX2100_CURSOR_YPOS;
				nReadMode	 		:= READ_MODE_BYTE;
				fbADSRead.DESTADDR 	:= ADR(nCursorPosY);
				fbADSRead.LEN		:= SIZEOF(nCursorPosY);
			3:
				(* CursorState *)
				nIndexOffset 		:= IOADS_IOF_CX2100_CURSOR;
				nReadMode			:= READ_MODE_BYTE;
				fbADSRead.DESTADDR 	:= ADR(nCursorMode);
				fbADSRead.LEN		:= SIZEOF(nCursorMode);
			END_CASE
		eCX2100_ReadBackLight:
			nIndexOffset 		:= IOADS_IOF_CX2100_BACKLIGHT_INT;
			nReadMode			:= READ_MODE_BYTE;
			fbADSRead.DESTADDR 	:= ADR(nBacklight);
			fbADSRead.LEN		:= SIZEOF(nBacklight);
		eCX2100_ReadLine1:
			(* Read Line1 *)
			nIndexOffset 		:= IOADS_IOF_CX2100_LINE1;
			nReadMode	 		:= READ_MODE_STRING;
			fbADSRead.DESTADDR 	:= ADR(sLine1);
			fbADSRead.LEN		:= SIZEOF(sLine1);
		eCX2100_ReadLine2:
			(* Read Line2 *)
			nIndexOffset 		:= IOADS_IOF_CX2100_LINE2;
			nReadMode	 		:= READ_MODE_STRING;
			fbADSRead.DESTADDR 	:= ADR(sLine2);
			fbADSRead.LEN		:= SIZEOF(sLine2);
		eCX2100_ReadLines:
			nReadStateMax := 2;
			IF NOT bStarted THEN
				nReadState := 1;
			END_IF
			CASE nReadState OF
			1:
				(* Read Line1 *)
				nIndexOffset 		:= IOADS_IOF_CX2100_LINE1;
				nReadMode	 		:= READ_MODE_STRING;
				fbADSRead.DESTADDR 	:= ADR(sLine1);
				fbADSRead.LEN		:= SIZEOF(sLine1);
			2:
				(* Read Line2 *)
				nIndexOffset 		:= IOADS_IOF_CX2100_LINE2;
				nReadMode			:= READ_MODE_STRING;
				fbADSRead.DESTADDR 	:= ADR(sLine2);
				fbADSRead.LEN		:= SIZEOF(sLine2);
			END_CASE
		END_CASE

		CASE nReadMode OF
			READ_MODE_IDLE :
				;
			READ_MODE_BYTE, READ_MODE_STRING:
				fbADSRead(
					NETID	:= sNetID,
					PORT	:= nPort,
					IDXGRP	:= IOADS_IOF_IGRP,
					IDXOFFS	:= nIndexOffset,
					READ	:= TRUE,
					TMOUT	:= t#1s
				);
		END_CASE;

		bStarted := TRUE;
		nState   := 1;
	END_IF

1:
	fbADSRead();
	IF NOT fbADSRead.BUSY OR (nReadMode = READ_MODE_IDLE) THEN
		IF fbADSRead.err THEN
			bError 		:= TRUE;
			nErrorID 	:= fbADSRead.ERRID;
		END_IF
		fbADSRead( READ:= FALSE );

		IF nReadState < nReadStateMax THEN
			(* read next object *)
			nReadState := nReadState + 1;
		ELSE
			(* done with reading *)
			bStarted 	:= FALSE;
			bBusy 		:= FALSE;
		END_IF

		nState := 0;
	END_IF
END_CASE
END_FUNCTION_BLOCK

(* POU FB_CXProfiler, ST *)
FUNCTION_BLOCK FB_CXProfiler
VAR_INPUT
	bStart					: BOOL;(*rising edge starts measurement and falling stops*)
	bReset					: BOOL;
END_VAR
VAR_OUTPUT
	bBusy					: BOOL;
	stData					: ST_CX_ProfilerStruct;
END_VAR
VAR CONSTANT
	iMAX_DATABUFF_SIZE		: INT := 100;
	iMAX_AVERAGE_MEASURES 	: INT := 100;
END_VAR
VAR
	fbRisingEdgeStart		: R_TRIG;
	fbRisingEdgeReset		: R_TRIG;
	fbFallingEdgeStart		: F_TRIG;
	fbGetCPUCounter			: GETCPUCOUNTER;
	dwOldCpuCntLo			: DWORD:=0;
	dwOldCpuCntHi			: DWORD:=0;
	dwOldCpuCntDiff			: DWORD:=0;
	dwNewCpuCntLo			: DWORD:=0;
	dwNewCpuCntHi			: DWORD:=0;
	dwNewCpuCntDiff		: DWORD:=0;
	aMeasureData			: ARRAY[0..iMAX_DATABUFF_SIZE] OF DWORD;
	dwTimeSum				: DWORD:=0;
	iMaxData					: UDINT:=1;
	iIdx							: DWORD:=0;
END_VAR
fbFallingEdgeStart(CLK:=bStart);

IF ( fbFallingEdgeStart.Q ) THEN
	fbGetCPUCounter();	(*get current counter value*)
	dwNewCpuCntLo := fbGetCPUCounter.cpuCntLoDW;
	dwNewCpuCntHi := fbGetCPUCounter.cpuCntHiDW;

	dwNewCpuCntDiff := F_CXSubTimeStamp(dwNewCpuCntLo, dwNewCpuCntHi, dwOldCpuCntLo, dwOldCpuCntHi);

	stData.dwLastExecTime	:=	 dwNewCpuCntDiff; (* in us *)

	(*calculate the min and max*)
	IF ( stData.dwMeasureCycle = 1 ) THEN  			(*first measurement*)
		stData.dwMinExecTime 	:= 	stData.dwLastExecTime;
		stData.dwMaxExecTime 	:= 	stData.dwLastExecTime;
	ELSE	(* ( Overflow->stData.MeasureCycle==0 ) or ( measure > 1 ) *)
		stData.dwMinExecTime 	:=	MIN( stData.dwMinExecTime, stData.dwLastExecTime );
		stData.dwMaxExecTime 	:=	MAX( stData.dwMaxExecTime, stData.dwLastExecTime );
	END_IF

	(* save last value to the data buffer *)
	aMeasureData[ stData.dwMeasureCycle MOD iMaxData  (*0..iMaxData - 1*)]	:= 	stData.dwLastExecTime;

	(*calculate average values*)
	dwTimeSum	:= 0;
	IF ( stData.dwMeasureCycle >= iMaxData ) OR ( stData.dwMeasureCycle = 0 ) THEN (*add all values*)
		FOR iIdx := 0 TO ( iMaxData - 1 ) DO
			dwTimeSum 	:= 	dwTimeSum + aMeasureData[ iIdx ];
		END_FOR
		stData.dwAverageExecTime	:= 	dwTimeSum / iMaxData;
	ELSE
		FOR  iIdx:=1  TO stData.dwMeasureCycle DO
			dwTimeSum 	:= 	dwTimeSum + aMeasureData[ iIdx ];
		END_FOR
		stData.dwAverageExecTime	:= 	dwTimeSum / stData.dwMeasureCycle;
	END_IF

	bBusy:=FALSE;
END_IF


fbRisingEdgeStart(CLK:=bStart);
fbRisingEdgeReset(CLK:=bReset);
IF ( fbRisingEdgeStart.Q ) THEN
	bBusy:=TRUE;

	IF ( fbRisingEdgeReset.Q ) THEN
		stData.dwLastExecTime := 0;
		stData.dwMinExecTime := 0;
		stData.dwMaxExecTime := 0;
		stData.dwAverageExecTime:=0;
		stData.dwMeasureCycle:=0;
		dwTimeSum := 0;
		FOR iIdx := 0 TO iMaxData DO
			aMeasureData[ iIdx ]:=0;	(*clear buffer*)
		END_FOR;
	END_IF

	iMaxData:= MAX( 2, MIN( iMAX_DATABUFF_SIZE,  iMAX_AVERAGE_MEASURES ) );
	stData.dwMeasureCycle	:=	stData.dwMeasureCycle + 1;		(*increment measure cycle counter*)

	fbGetCPUCounter();								(*get current counter value*)
													(* save start  value*)
	dwOldCpuCntLo := fbGetCPUCounter.cpuCntLoDW;
	dwOldCpuCntHi := fbGetCPUCounter.cpuCntHiDW;
END_IF
END_FUNCTION_BLOCK

(* POU FB_CXSetTextDisplay, ST *)
FUNCTION_BLOCK FB_CXSetTextDisplay
VAR_INPUT
	bExecute 		: BOOL;
	nDevID			: UDINT;
	nMode			: E_CX1100_DisplayModes;
	stLine 			: STRING(20);
	nCursorPos 		: DWORD;
END_VAR
VAR_OUTPUT
	bBusy 			: BOOL;
	bErr			: BOOL;
	nErrorID		: UDINT;
END_VAR
VAR
	step 			: INT := 100;
	fbADSWrite 		: ADSWRITE;
	bStarted 		: BOOL;
	nIndexOffset	: UDINT;
	nWriteMode 		: INT;
	fbOnTrigger		: R_TRIG;
	temp 			: DWORD;
END_VAR
VAR CONSTANT
	(* write mode *)
	WRITE_MODE_IDLE		: INT := 1;
	WRITE_MODE_BYTE		: INT := 2;
	WRITE_MODE_STRING	: INT := 3;

	(*  CX1100 *)
	IOADS_IOF_CX1100_WRITE1LINE 	: UDINT :=	16#FFFF00FF;
	IOADS_IOF_CX1100_WRITE2LINE 	: UDINT :=	16#FFFF40FF;
	IOADS_IOF_CX1100_WRITECURSOR 	: UDINT :=	16#FFFF80FF;
	IOADS_IOF_CX1100_FILLRAW 		: UDINT :=	16#FFFF81FF;
	IOADS_IOF_CX1100_CURSOR_OFF 	: UDINT :=	16#FFFF90FF;
	IOADS_IOF_CX1100_CURSOR_ON 		: UDINT :=	16#FFFF91FF;
	IOADS_IOF_CX1100_CURSOR_BOFF 	: UDINT :=	16#FFFF92FF;
	IOADS_IOF_CX1100_CURSOR_BON 	: UDINT :=	16#FFFF93FF;
	IOADS_IOF_CX1100_DISPLAY_OFF 	: UDINT :=	16#FFFF94FF;
	IOADS_IOF_CX1100_DISPLAY_ON 	: UDINT :=	16#FFFF95FF;
	IOADS_IOF_CX1100_BACKLIGHT_ON 	: UDINT :=	16#FFFF96FF;
	IOADS_IOF_CX1100_BACKLIGHT_OFF 	: UDINT :=	16#FFFF97FF;
	IOADS_IOF_CX1100_CLEARDISPLAY 	: UDINT :=	16#FFFFA0FF;

	IOADS_IOF_CX1100_TERMTYPES 		: UDINT :=	16#FFFF0001;
END_VAR
CASE step OF
100 :
	fbOnTrigger(CLK:= bExecute);
    IF fbOnTrigger.Q OR bStarted
	THEN
		bStarted := TRUE;
		bBusy := TRUE;
		bErr := FALSE;
		nErrorID := 0;
		(* select action *)
		CASE nMode OF
			e_CX1100_DisplayNoAction:
				nIndexOffset := 0;
				nWriteMode 	 := WRITE_MODE_IDLE;
			e_CX1100_DisplayOn:
				nIndexOffset := IOADS_IOF_CX1100_DISPLAY_ON;
				nWriteMode	 := WRITE_MODE_BYTE;
			e_CX1100_DisplayOff:
				nIndexOffset := IOADS_IOF_CX1100_DISPLAY_OFF;
				nWriteMode	 := WRITE_MODE_BYTE;
			e_CX1100_CursorOn:
				nIndexOffset := IOADS_IOF_CX1100_CURSOR_ON;
				nWriteMode	 := WRITE_MODE_BYTE;
			e_CX1100_CursorOff:
				nIndexOffset := IOADS_IOF_CX1100_CURSOR_OFF;
				nWriteMode	 := WRITE_MODE_BYTE;
			e_CX1100_CursorBlinkOn:
				nIndexOffset := IOADS_IOF_CX1100_CURSOR_BON;
				nWriteMode	 := WRITE_MODE_BYTE;
			e_CX1100_CursorBlinkOff:
				nIndexOffset := IOADS_IOF_CX1100_CURSOR_BOFF;
				nWriteMode	 := WRITE_MODE_BYTE;
			e_CX1100_BackLightOn:
				nIndexOffset := IOADS_IOF_CX1100_BACKLIGHT_ON;
				nWriteMode	 := WRITE_MODE_BYTE;
			e_CX1100_BackLightOff:
				nIndexOffset := IOADS_IOF_CX1100_BACKLIGHT_OFF;
				nWriteMode	 := WRITE_MODE_BYTE;
			e_CX1100_ClearDisplay:
				nIndexOffset := IOADS_IOF_CX1100_CLEARDISPLAY;
				nWriteMode	 := WRITE_MODE_BYTE;
			e_CX1100_WriteLine1:
				IF nCursorPos <> 0
				THEN
					IF nCursorPos < 15
					THEN
						nIndexOffset := DWORD_TO_UDINT( UDINT_TO_DWORD(IOADS_IOF_CX1100_WRITE1LINE) OR (SHL(nCursorPos,8)));
					ELSE
						nIndexOffset := 0;
						nWriteMode	 := WRITE_MODE_IDLE;
						bErr := TRUE;
						nErrorID := 4711;
					END_IF;
				ELSE
					nIndexOffset := IOADS_IOF_CX1100_WRITE1LINE;
				END_IF;
				nWriteMode := WRITE_MODE_STRING;
			e_CX1100_WriteLine2:
				IF nCursorPos <> 0
				THEN
					IF nCursorPos < 15
					THEN
						nIndexOffset := DWORD_TO_UDINT( UDINT_TO_DWORD(IOADS_IOF_CX1100_WRITE2LINE) OR (SHL(nCursorPos,8)));
					ELSE
						nIndexOffset := 0;
						nWriteMode	 := WRITE_MODE_IDLE;
						bErr := TRUE;
						nErrorID := 4711;
					END_IF;
				ELSE
					nIndexOffset := IOADS_IOF_CX1100_WRITE2LINE;
				END_IF;
				nWriteMode := WRITE_MODE_STRING;
		ELSE
			;
		END_CASE;

		CASE nWriteMode OF
			WRITE_MODE_IDLE :
				;
			WRITE_MODE_BYTE:
				fbADSWrite(NETID:= '',
					PORT	:= 300,
					IDXGRP	:= IOADS_IGR_IODEVICESTATE_BASE+nDevID,
					IDXOFFS	:= nIndexOffset,
					LEN		:= 0,
					SRCADDR:= 0,
					WRITE	:= TRUE,
					TMOUT	:= t#1s);
			WRITE_MODE_STRING:
				fbADSWrite(NETID:= '',
					PORT	:= 300,
					IDXGRP	:= IOADS_IGR_IODEVICESTATE_BASE+nDevID,
					IDXOFFS	:= nIndexOffset,
					LEN		:= LEN(stLine),
					SRCADDR	:= ADR(stLine),
					WRITE	:= TRUE,
					TMOUT	:= t#1s);
		END_CASE;

		IF NOT fbADSWrite.BUSY OR (nWriteMode = WRITE_MODE_IDLE)
		THEN
			bStarted := FALSE;
			step := 300;
		END_IF;
	END_IF;
300:
	IF NOT fbADSWrite.err
	THEN
		step := 100;
	ELSE
		bErr := TRUE;
		nErrorID := fbADSWrite.ERRID;
		step := 100;
	END_IF;
	fbADSWrite( WRITE:= FALSE );
	bBusy := FALSE;
END_CASE;
END_FUNCTION_BLOCK

(* POU FB_CXSetTextDisplayUSB, ST *)
FUNCTION_BLOCK FB_CXSetTextDisplayUSB
VAR_INPUT
	bExecute		: BOOL;
	sNetID			: T_AmsNetID;
	nPort			: T_AmsPort;
	eMode			: E_CX2100_DisplayModesWr;
	sLine1			: STRING;
	sLine2			: STRING;
	nCursorPosX		: USINT;
	nCursorPosY		: USINT;
END_VAR
VAR_OUTPUT
	bBusy 			: BOOL;
	bError			: BOOL;
	nErrorID		: UDINT;
END_VAR
{library private}
VAR
	eModeAct		: E_CX2100_DisplayModesWr;
	nState 			: INT := 0;
	bStarted 		: BOOL;
	fbOnTrigger		: R_TRIG;
	fbADSWrite 		: ADSWRITE;
	nIndexOffset	: UDINT;
	nWriteMode 		: INT;
	nCursorMode		: USINT;
	nBackLightVal	: USINT;
	nWriteState		: INT;
	nWriteStateMax	: INT;
	sClearLine 		: STRING := '';
END_VAR
VAR CONSTANT
	(* write mode *)
	WRITE_MODE_IDLE		: INT := 1;
	WRITE_MODE_BYTE		: INT := 2;
	WRITE_MODE_STRING	: INT := 3;

	(* CX1200*)
	IOADS_IOF_CX2100_BACKLIGHT_INT 	: UDINT :=	16#80000011; (* backlight 0..255 *)
	IOADS_IOF_CX2100_LINE1 			: UDINT :=	16#80080011; (* read/write line 1 *)
	IOADS_IOF_CX2100_LINE2		 	: UDINT :=	16#80080012; (* read/write line 2 *)
	IOADS_IOF_CX2100_CURSOR		 	: UDINT :=	16#80080019; (* cursor ... 0 Off; 1 On; 2 Blink *)
	IOADS_IOF_CX2100_CURSOR_XPOS 	: UDINT :=	16#8008001A; (* cursor position in X *)
	IOADS_IOF_CX2100_CURSOR_YPOS 	: UDINT :=	16#8008001B; (* cursor position in Y *)
	IOADS_IOF_IGRP					: UDINT	:= 16#F302;		(* ADS index group OF the CX2100 mailbox *)
END_VAR
{library public}
CASE nState OF
0 :
	fbOnTrigger(CLK:= bExecute);
    IF fbOnTrigger.Q OR bStarted THEN
		(* initialize command *)
		IF NOT bStarted THEN
			bBusy 			:= TRUE;
			bError 			:= FALSE;
			nErrorID 		:= 0;
			eModeAct 		:= eMode;
			nWriteState		:= 0;
			nWriteStateMax	:= 0;
		END_IF

		(* select action *)
		CASE eModeAct OF
			eCX2100_DisplayNoActionWr:
				nIndexOffset 		:= 0;
				nWriteMode 	 		:= WRITE_MODE_IDLE;
			eCX2100_CursorOn:
				nIndexOffset 		:= IOADS_IOF_CX2100_CURSOR;
				nWriteMode	 		:= WRITE_MODE_BYTE;
				nCursorMode	 		:= 1;
				fbADSWrite.SRCADDR 	:= ADR(nCursorMode);
				fbADSWrite.LEN 		:= SIZEOF(nCursorMode);
			eCX2100_CursorOff:
				nIndexOffset 		:= IOADS_IOF_CX2100_CURSOR;
				nWriteMode	 		:= WRITE_MODE_BYTE;
				nCursorMode	 		:= 0;
				fbADSWrite.SRCADDR 	:= ADR(nCursorMode);
				fbADSWrite.LEN 		:= SIZEOF(nCursorMode);
			eCX2100_CursorBlinkOn:
				nIndexOffset 		:= IOADS_IOF_CX2100_CURSOR;
				nWriteMode	 		:= WRITE_MODE_BYTE;
				nCursorMode	 		:= 2;
				fbADSWrite.SRCADDR 	:= ADR(nCursorMode);
				fbADSWrite.LEN 		:= SIZEOF(nCursorMode);
			eCX2100_CursorBlinkOff:
				nIndexOffset 		:= IOADS_IOF_CX2100_CURSOR;
				nWriteMode	 		:= WRITE_MODE_BYTE;
				nCursorMode	 		:= 0;
				fbADSWrite.SRCADDR 	:= ADR(nCursorMode);
				fbADSWrite.LEN 		:= SIZEOF(nCursorMode);
			eCX2100_BackLightOn:
				nIndexOffset 		:= IOADS_IOF_CX2100_BACKLIGHT_INT;
				nWriteMode	 		:= WRITE_MODE_BYTE;
				nBackLightVal		:= 255;
				fbADSWrite.SRCADDR 	:= ADR(nBackLightVal);
				fbADSWrite.LEN 		:= SIZEOF(nBackLightVal);
			eCX2100_BackLightOff:
				nIndexOffset 		:= IOADS_IOF_CX2100_BACKLIGHT_INT;
				nWriteMode	 		:= WRITE_MODE_BYTE;
				nBackLightVal		:= 0;
				fbADSWrite.SRCADDR 	:= ADR(nBackLightVal);
				fbADSWrite.LEN 		:= SIZEOF(nBackLightVal);
			eCX2100_CursorPosX:
				nIndexOffset 		:= IOADS_IOF_CX2100_CURSOR_XPOS;
				nWriteMode	 		:= WRITE_MODE_BYTE;
				fbADSWrite.SRCADDR 	:= ADR(nCursorPosX);
				fbADSWrite.LEN 		:= SIZEOF(nCursorPosX);
			eCX2100_CursorPosY:
				nIndexOffset 		:= IOADS_IOF_CX2100_CURSOR_YPOS;
				nWriteMode	 		:= WRITE_MODE_BYTE;
				fbADSWrite.SRCADDR 	:= ADR(nCursorPosY);
				fbADSWrite.LEN 		:= SIZEOF(nCursorPosY);
			eCX2100_CursorPosXY:
				nWriteStateMax := 2;
				IF NOT bStarted THEN
					nWriteState := 1;
				END_IF
				CASE nWriteState OF
				1:
					(* CursorPosX *)
					nIndexOffset 		:= IOADS_IOF_CX2100_CURSOR_XPOS;
					nWriteMode	 		:= WRITE_MODE_BYTE;
					fbADSWrite.SRCADDR 	:= ADR(nCursorPosX);
					fbADSWrite.LEN 		:= SIZEOF(nCursorPosX);
				2:
					(* CursorPosY *)
					nIndexOffset 		:= IOADS_IOF_CX2100_CURSOR_YPOS;
					nWriteMode	 		:= WRITE_MODE_BYTE;
					fbADSWrite.SRCADDR 	:= ADR(nCursorPosY);
					fbADSWrite.LEN 		:= SIZEOF(nCursorPosY);
				END_CASE
			eCX2100_ClearDisplay:
				nWriteStateMax := 2;
				IF NOT bStarted THEN
					nWriteState := 1;
				END_IF
				CASE nWriteState OF
				1:
					(* Write Line1 *)
					nIndexOffset 		:= IOADS_IOF_CX2100_LINE1;
					nWriteMode	 		:= WRITE_MODE_STRING;
					fbADSWrite.SRCADDR 	:= ADR(sClearLine);
					fbADSWrite.LEN 		:= SIZEOF(sClearLine);
				2:
					(* Write Line2 *)
					nIndexOffset 		:= IOADS_IOF_CX2100_LINE2;
					nWriteMode	 		:= WRITE_MODE_STRING;
					fbADSWrite.SRCADDR 	:= ADR(sClearLine);
					fbADSWrite.LEN 		:= SIZEOF(sClearLine);
				END_CASE
			eCX2100_WriteLine1:
				(* Write Line1 *)
				nIndexOffset 		:= IOADS_IOF_CX2100_LINE1;
				nWriteMode	 		:= WRITE_MODE_STRING;
				fbADSWrite.SRCADDR 	:= ADR(sLine1);
				fbADSWrite.LEN 		:= SIZEOF(sLine1);
			eCX2100_WriteLine2:
				(* Write Line2 *)
				nIndexOffset 		:= IOADS_IOF_CX2100_LINE2;
				nWriteMode	 		:= WRITE_MODE_STRING;
				fbADSWrite.SRCADDR 	:= ADR(sLine2);
				fbADSWrite.LEN 		:= SIZEOF(sLine2);
			eCX2100_WriteLines:
				nWriteStateMax := 2;
				IF NOT bStarted THEN
					nWriteState := 1;
				END_IF
				CASE nWriteState OF
				1:
					(* Write Line1 *)
					nIndexOffset 		:= IOADS_IOF_CX2100_LINE1;
					nWriteMode	 		:= WRITE_MODE_STRING;
					fbADSWrite.SRCADDR 	:= ADR(sLine1);
					fbADSWrite.LEN 		:= SIZEOF(sLine1);
				2:
					(* Write Line2 *)
					nIndexOffset 		:= IOADS_IOF_CX2100_LINE2;
					nWriteMode	 		:= WRITE_MODE_STRING;
					fbADSWrite.SRCADDR 	:= ADR(sLine2);
					fbADSWrite.LEN 		:= SIZEOF(sLine2);
				END_CASE

		ELSE
			;
		END_CASE

		CASE nWriteMode OF
			WRITE_MODE_IDLE :
				;
			WRITE_MODE_BYTE, WRITE_MODE_STRING:
				fbADSWrite(
					NETID	:= sNetID,
					PORT	:= nPort,
					IDXGRP	:= IOADS_IOF_IGRP,
					IDXOFFS	:= nIndexOffset,
					WRITE	:= TRUE,
					TMOUT	:= t#1s
				);
		END_CASE;

		bStarted := TRUE;
		nState   := 1;
	END_IF

1:
	fbADSWrite();
	IF NOT fbADSWrite.BUSY OR (nWriteMode = WRITE_MODE_IDLE) THEN
		IF fbADSWrite.err THEN
			bError 		:= TRUE;
			nErrorID 	:= fbADSWrite.ERRID;
		END_IF
		fbADSWrite( WRITE:= FALSE );

		IF nWriteState < nWriteStateMax THEN
			(* write next object *)
			nWriteState := nWriteState + 1;
		ELSE
			(* done with writing *)
			bStarted := FALSE;
			bBusy := FALSE;
		END_IF

		nState := 0;
	END_IF
END_CASE
END_FUNCTION_BLOCK

(* POU FB_CXSimpleUps, ST *)
FUNCTION_BLOCK FB_CXSimpleUps
VAR_INPUT
	bDIPDisable			: BOOL;	(* If TRUE override Dip Switch *)
	iDischargeLevel		: USINT;(* Discharge Switch Off Level: 0 = 100%, 9 = 90%, 8 = 80%, ..., 2 = 20%, 1 = 10% *)
	tDelay				: TIME;	(* Time to hold during power failure (shutdown after timer ellapses) [0.5s .. 10s] *)
END_VAR
VAR_OUTPUT
	bPowerFailure		: BOOL;	(* True if power fault detected *)
	bShutdownActive		: BOOL;	(* True if shutdown is actively executed *)
	bUpsReady			: BOOL;	(* True if UPS 24V Out is OK *)
	b24VInOK			: BOOL;	(* True if UPS 24V In is OK *)
	bHolding			: BOOL;	(* True if power fault detected and tDelay not yet ellapsed *)
	tTimeUntilShutdown	: TIME;	(* Remaining Time until system shuts down during power failure *)
	eUpsState			: E_UPS_STATE; (* UPS-State [UNDEF | CHARGING | CHARGED | DISCHARGE |
													 DISCHARGE_RESTART | OUTPUT_OFF | OVERLOAD] *)
END_VAR
VAR
	Ii24VState AT %I* 	: BYTE;
	IiChargeState AT %I*: BYTE;
	QiControl AT %Q*	: BYTE := 2#0000_1000; (* set bit 3 - auto reset *)
	QiDipControl AT %Q*	: BYTE;

	iState				: INT := 0; (* 0: IDLE, 1: HOLDING, 2: SHUTDOWN *)
	HoldTimer			: TON;
	fbShutdown			: ADSWRTCTL;  (* Windows shutdown *)
	dwDelay				: DWORD := 0; (* 0 immediate shutdown of Windows, [s] *)
	WaitStateTime		: TON;		(*Wait for state UPS*)
	DischargeTime		: TON;		(*Catch state UPS discharging-restart *)
	bEndOfHolding		: BOOL;		(*Phase before Shutdown activ*)
END_VAR
VAR CONSTANT
	tWaitStateTime		: TIME := t#2s500ms;
	tDischargeTime		: TIME := t#2s500ms;
END_VAR
(* status *)
b24VInOK		:= Ii24VState.1;
bUpsReady		:= Ii24VState.0;
bPowerFailure 	:= NOT(Ii24VState.1);
eUpsState		:= SHR((Ii24VState AND 16#F0), 4);
QiControl.2 	:= bDIPDisable;

(* limit holding time *)
IF tDelay < T#500ms THEN
	tDelay := T#500ms;
ELSIF tDelay > T#10s THEN
	tDelay := T#10s;
END_IF

HoldTimer(PT := tDelay + T#1s100ms, IN := bPowerFailure);
WaitStateTime(PT := tWaitStateTime, IN := bEndOfHolding);
DischargeTime(PT := tDischargeTime, IN := ((eUpsState = eUPS_DISCHARGE_RESTART) AND b24VInOK));

(* override DIP switch with iDischargeLevel *)
IF bDIPDisable THEN
	IF iDischargeLevel > 9 THEN  (* limit SW Dip Switch *)
		QiDipControl := 0;
	ELSE
		QiDipControl := iDischargeLevel;
	END_IF
END_IF

CASE iState OF
0: (* IDLE *)
	(* make sure link to IiChargeState exists (assume link to Ii24VState is then also there) before evaluating power failure to avoid constant reboot *)
	QiControl.3 := TRUE; (* alway set auto reset *)

	IF bPowerFailure AND (eUpsState <> eUPS_UNDEF) THEN
		(* hold on power failure power failure*)
		iState 		:= 1;
	ELSIF DischargeTime.Q THEN
		(* catch longer period of discharging despite no power failure *)
		bEndOfHolding	:= TRUE;
		QiControl.3 	:= FALSE; (* clear auto reset *)
		iState 			:= 2;
	END_IF

1: (* HOLD *)
	IF b24VInOK THEN
		(* power failure has ended before hold timer ellapsed *)
		iState 		:= 0;

	ELSIF HoldTimer.Q THEN
		(* power failure has continued until hold timer ellapsed *)
		bEndOfHolding	:= TRUE;
		QiControl.3 	:= FALSE; (* clear auto reset *)
		iState 			:= 2;
	END_IF

2: (* Wait for state UPS *)
	IF WaitStateTime.Q  THEN
		bEndOfHolding	:= FALSE;
		IF (eUpsState <> eUPS_DISCHARGE_RESTART) AND (eUpsState <> eUPS_DISCHARGE) THEN
			(* no shutdown required since CX power supply is not discharging-restart *)
			iState := 0;
			QiControl.3 := TRUE; (* alway set auto reset *)
		ELSE
			(* shutdown required since CX power supply is discharging-restart *)
			bShutdownActive := TRUE;
			fbShutdown(
				NETID 		:= '',
				PORT 		:= AMSPORT_R3_SYSSERV,
				ADSSTATE 	:= ADSSTATE_POWERFAILURE, (* Windows Shutdown *)
				DEVSTATE 	:= 0,
				LEN 		:= SIZEOF(dwDelay),
				SRCADDR 	:= ADR(dwDelay),
				Write 		:= TRUE,
				TMOUT 	:= T#3s
			);
			iState 			:= 3;
		END_IF
	END_IF

3: (* SHUTDOWN *)
	fbShutdown(Write := TRUE);
END_CASE

(* status *)
bHolding 			:= QiControl.3 AND bPowerFailure;
tTimeUntilShutdown	:= HoldTimer.PT - HoldTimer.ET;
END_FUNCTION_BLOCK
